FUNCTION_BLOCK LibrariesAndReusableCode
VAR_INPUT
	Number : REAL;
END_VAR
VAR_OUTPUT
END_VAR
VAR
	 
END_VAR

// absolute value
IF Number < 0 THEN 
	Number := Number*(-1); 
ELSE
	Number := Number ; 
END_IF

Number := ABS(Number);

END_FUNCTION_BLOCK

(* stored: Version 1.1.0.1
   POU LibrariesAndReusableCode: Id {38099b21-d6f0-4ff4-bfb0-c8ab3f6f1202}, SpecialFunc None *)
